PROGRAM P_Demo_FB_JsonSaxWriter_AddUlint
VAR
    fbParser : FB_JsonSaxWriter; // 父 FB 实例
    value : ULINT;
    bTrigger : BOOL := FALSE; // 在线置 TRUE 触发一次调用
    bTriggerPrev : BOOL;
END_VAR

// =============================================================================
// 场景：SAX 流式生成 JSON 时追加 Ulint 类型的值/键值对。
// 价值：无 DOM 中间态，内存最省、速度最快。
// 验证：登录 PLC 在线写 bTrigger := TRUE 触发，monitor 返回值/输出参数。具体步骤见下方注释。
// 验证步骤：
//   1. 右键 PLC 项目下 POUs 文件夹 → Add → Existing Item → 选本 .TcPOU 文件
//   2. 引用 Tc3_JsonXml（References → Add library）
//   3. 编译 → 登录 → 运行；按 verify 注释里给出的在线写值操作
// =============================================================================

// 上升沿触发一次方法调用并观察输出。
IF bTrigger AND NOT bTriggerPrev THEN
    fbParser.AddUlint(
        value := value
    );
END_IF;
bTriggerPrev := bTrigger;

END_PROGRAM

(* stored: Version 1.1.0.1, ProductVersion 3.1.4024.5
   POU P_Demo_FB_JsonSaxWriter_AddUlint: Id {9353c96c-313e-5df8-9edc-f34e4a453ad2}, SpecialFunc None *)
